FUNCTION_BLOCK CU040ExampleCompositComponent EXTENDS TcoCore.TcoComponent
VAR_INPUT
END_VAR
VAR_OUTPUT
END_VAR
VAR
END_VAR

END_FUNCTION_BLOCK

(* stored: Version 1.1.0.1
   POU CU040ExampleCompositComponent: Id {3c5e4a79-8f8d-4e5e-acac-5d013d7f251e}, SpecialFunc None *)
